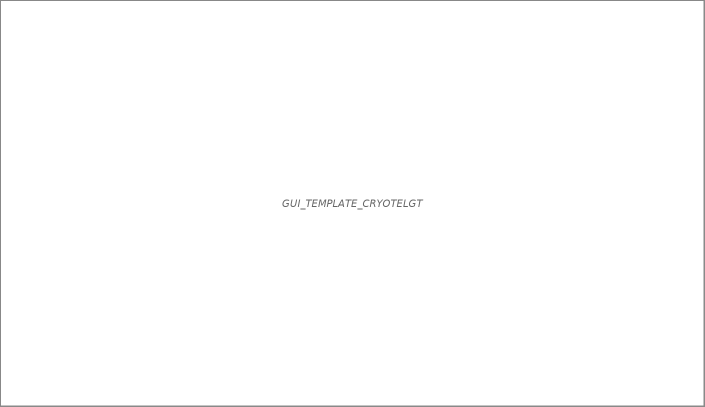
VISUALIZATION GUI_CRYOTELGT  // 705x407
    Frame (0,0 705x407)
        shows GUI_TEMPLATE_CRYOTELGT(m_Instance := MAIN.cooler, m_bEnable := MAIN.bEnable_cooler)
END_VISUALIZATION

(* stored: Version 1.1.0.1, ProductVersion 3.1.4024.12
   Visu GUI_CRYOTELGT: Id {a388866c-9f55-4c03-8700-778ac11822f0} *)
